_CFC_ (* Continuous Function Chart, elements in execution order *)
#0 TON_KV:TON(IN: NOT SCHU_P2_3_KV1_DI4, PT: T#5s)
#1 RS_Net_vhk_napr:SR(SET1: #0.Q, RESET: SCHU_P2_3_SB)
#2 SCHU_P2_3_Z_NET_VH_NAPR <= #1.Q1
_END_CFC_
(* the same logic as Structured Text *)
TON_KV(IN := NOT SCHU_P2_3_KV1_DI4, PT := T#5s);
RS_Net_vhk_napr(SET1 := TON_KV.Q, RESET := SCHU_P2_3_SB);
SCHU_P2_3_Z_NET_VH_NAPR := RS_Net_vhk_napr.Q1;
END_PROGRAM

(* POU TZBiS/TZB/Z_NP, CFC *)
PROGRAM Z_NP
VAR
	TON_PDS2: TON;
	TON_ReRab: TON;
	TON_MVKL: TON;
	TON_AVT: TON;
	TP_SR: TP;
	SR_NP_M1: SR;
	SR_NP_M2: SR;
	TON_MVKL_M1: TON;
	TON_AVT_M1: TON;
	TON_AVT_M2: TON;
	TON_MVKL_M2: TON;
END_VAR
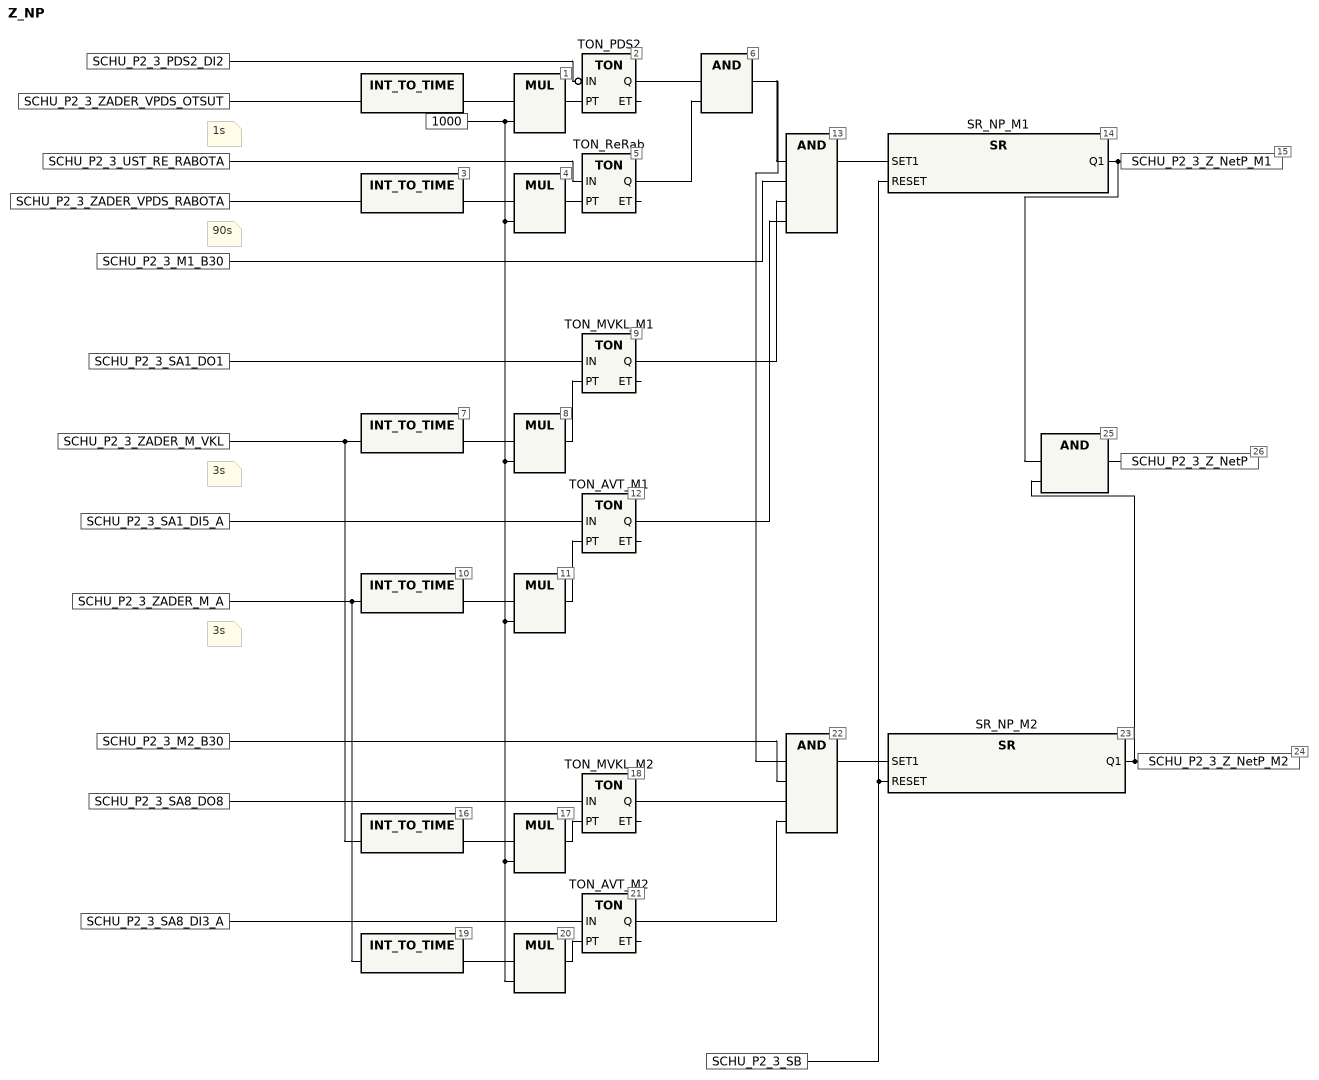
_CFC_ (* Continuous Function Chart, elements in execution order *)
(* 1s *)
(* 90s *)
(* 3s *)
(* 3s *)
#0 INT_TO_TIME(SCHU_P2_3_ZADER_VPDS_OTSUT)
#1 MUL(#0, 1000)
#2 TON_PDS2:TON(IN: NOT SCHU_P2_3_PDS2_DI2, PT: #1)
#3 INT_TO_TIME(SCHU_P2_3_ZADER_VPDS_RABOTA)
#4 MUL(#3, 1000)
#5 TON_ReRab:TON(IN: SCHU_P2_3_UST_RE_RABOTA, PT: #4)
#6 AND(#2.Q, #5.Q)
#7 INT_TO_TIME(SCHU_P2_3_ZADER_M_VKL)
#8 MUL(#7, 1000)
#9 TON_MVKL_M1:TON(IN: SCHU_P2_3_SA1_DO1, PT: #8)
#10 INT_TO_TIME(SCHU_P2_3_ZADER_M_A)
#11 MUL(#10, 1000)
#12 TON_AVT_M1:TON(IN: SCHU_P2_3_SA1_DI5_A, PT: #11)
#13 AND(#6, SCHU_P2_3_M1_B30, #9.Q, #12.Q)
#14 SR_NP_M1:SR(SET1: #13, RESET: SCHU_P2_3_SB)
#15 SCHU_P2_3_Z_NetP_M1 <= #14.Q1
#16 INT_TO_TIME(SCHU_P2_3_ZADER_M_VKL)
#17 MUL(#16, 1000)
#18 TON_MVKL_M2:TON(IN: SCHU_P2_3_SA8_DO8, PT: #17)
#19 INT_TO_TIME(SCHU_P2_3_ZADER_M_A)
#20 MUL(#19, 1000)
#21 TON_AVT_M2:TON(IN: SCHU_P2_3_SA8_DI3_A, PT: #20)
#22 AND(#6, SCHU_P2_3_M2_B30, #18.Q, #21.Q)
#23 SR_NP_M2:SR(SET1: #22, RESET: SCHU_P2_3_SB)
#24 SCHU_P2_3_Z_NetP_M2 <= #23.Q1
#25 AND(#14.Q1, #23.Q1)
#26 SCHU_P2_3_Z_NetP <= #25
_END_CFC_
(* the same logic as Structured Text *)
(* 1s *)
(* 90s *)
(* 3s *)
(* 3s *)
TON_PDS2(IN := NOT SCHU_P2_3_PDS2_DI2, PT := INT_TO_TIME(SCHU_P2_3_ZADER_VPDS_OTSUT) * 1000);
TON_ReRab(IN := SCHU_P2_3_UST_RE_RABOTA, PT := INT_TO_TIME(SCHU_P2_3_ZADER_VPDS_RABOTA) * 1000);
TON_MVKL_M1(IN := SCHU_P2_3_SA1_DO1, PT := INT_TO_TIME(SCHU_P2_3_ZADER_M_VKL) * 1000);
TON_AVT_M1(IN := SCHU_P2_3_SA1_DI5_A, PT := INT_TO_TIME(SCHU_P2_3_ZADER_M_A) * 1000);
SR_NP_M1(SET1 := (TON_PDS2.Q AND TON_ReRab.Q) AND SCHU_P2_3_M1_B30 AND TON_MVKL_M1.Q AND TON_AVT_M1.Q, RESET := SCHU_P2_3_SB);
SCHU_P2_3_Z_NetP_M1 := SR_NP_M1.Q1;
TON_MVKL_M2(IN := SCHU_P2_3_SA8_DO8, PT := INT_TO_TIME(SCHU_P2_3_ZADER_M_VKL) * 1000);
TON_AVT_M2(IN := SCHU_P2_3_SA8_DI3_A, PT := INT_TO_TIME(SCHU_P2_3_ZADER_M_A) * 1000);
SR_NP_M2(SET1 := (TON_PDS2.Q AND TON_ReRab.Q) AND SCHU_P2_3_M2_B30 AND TON_MVKL_M2.Q AND TON_AVT_M2.Q, RESET := SCHU_P2_3_SB);
SCHU_P2_3_Z_NetP_M2 := SR_NP_M2.Q1;
SCHU_P2_3_Z_NetP := SR_NP_M1.Q1 AND SR_NP_M2.Q1;
END_PROGRAM

(* POU TZBiS/TZB/Z_OTKAZ_VTOR_ZEP, CFC *)
PROGRAM Z_OTKAZ_VTOR_ZEP
VAR
	rs_otkaz_vtor_sep: RS;
END_VAR
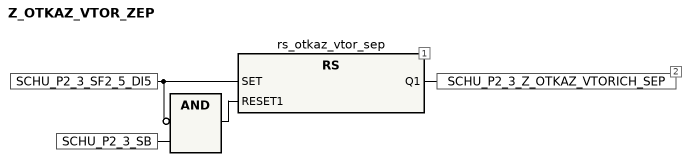
_CFC_ (* Continuous Function Chart, elements in execution order *)
#0 AND(NOT SCHU_P2_3_SF2_5_DI5, SCHU_P2_3_SB)
#1 rs_otkaz_vtor_sep:RS(SET: SCHU_P2_3_SF2_5_DI5, RESET1: #0)
#2 SCHU_P2_3_Z_OTKAZ_VTORICH_SEP <= #1.Q1
_END_CFC_
(* the same logic as Structured Text *)
rs_otkaz_vtor_sep(SET := SCHU_P2_3_SF2_5_DI5, RESET1 := NOT SCHU_P2_3_SF2_5_DI5 AND SCHU_P2_3_SB);
SCHU_P2_3_Z_OTKAZ_VTORICH_SEP := rs_otkaz_vtor_sep.Q1;
END_PROGRAM

(* POU TZBiS/TZB/Z_P1_NP, CFC *)
PROGRAM Z_P1_NP
VAR
	SR_P1_NPit: SR;
END_VAR
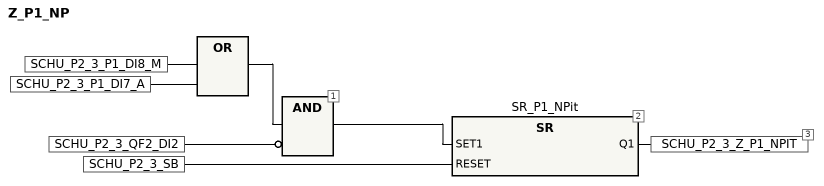
_CFC_ (* Continuous Function Chart, elements in execution order *)
#0 OR(SCHU_P2_3_P1_DI8_M, SCHU_P2_3_P1_DI7_A)
#1 AND(#0, NOT SCHU_P2_3_QF2_DI2)
#2 SR_P1_NPit:SR(SET1: #1, RESET: SCHU_P2_3_SB)
#3 SCHU_P2_3_Z_P1_NPIT <= #2.Q1
_END_CFC_
(* the same logic as Structured Text *)
SR_P1_NPit(SET1 := (SCHU_P2_3_P1_DI8_M OR SCHU_P2_3_P1_DI7_A) AND NOT SCHU_P2_3_QF2_DI2, RESET := SCHU_P2_3_SB);
SCHU_P2_3_Z_P1_NPIT := SR_P1_NPit.Q1;
END_PROGRAM

(* POU TZBiS/TZB/Z_P2_NP, CFC *)
PROGRAM Z_P2_NP
VAR
	SR_P2_NPit: SR;
END_VAR
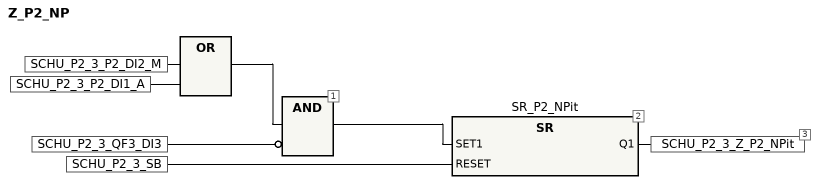
_CFC_ (* Continuous Function Chart, elements in execution order *)
#0 OR(SCHU_P2_3_P2_DI2_M, SCHU_P2_3_P2_DI1_A)
#1 AND(#0, NOT SCHU_P2_3_QF3_DI3)
#2 SR_P2_NPit:SR(SET1: #1, RESET: SCHU_P2_3_SB)
#3 SCHU_P2_3_Z_P2_NPit <= #2.Q1
_END_CFC_
(* the same logic as Structured Text *)
SR_P2_NPit(SET1 := (SCHU_P2_3_P2_DI2_M OR SCHU_P2_3_P2_DI1_A) AND NOT SCHU_P2_3_QF3_DI3, RESET := SCHU_P2_3_SB);
SCHU_P2_3_Z_P2_NPit := SR_P2_NPit.Q1;
END_PROGRAM

(* POU TZBiS/TZB/Z_P2_Otk, CFC *)
PROGRAM Z_P2_Otk
VAR
	SR_P2_Otkaz: SR;
	UE2_VL_Old: REAL;
	TON_UE2: TON;
	RT_P2_RUN: R_TRIG;
END_VAR
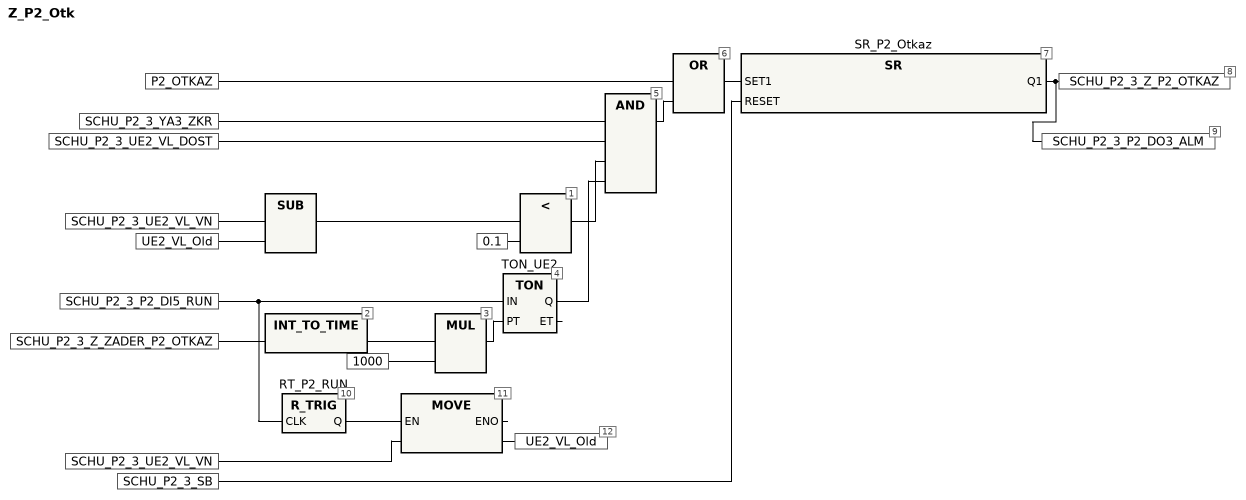
